// TwinCAT 3 PLC project PRG_B_MachineControl
// Title: B_MachineControl
// Company: RafalOS
// Author: Rafał Osajda
// ProjectVersion: 0.0.0.1
// ProgramVersion: 3.1.4024.0
// libraries:
//   B_Base, * (RafalOS)
//   B_IO, * (RafalOS)
//   Tc2_Standard, * (Beckhoff Automation GmbH)
//   Tc2_System, * (Beckhoff Automation GmbH)
//   Tc3_Module, * (Beckhoff Automation GmbH)
// project tree:
//   DUTs/ ST_Safety.TcDUT, ST_SafetyGroupStates.TcDUT
//   GVLs/ GVL_MCIO.TcGVL, GVL_MCConstans.TcGVL
//   / PlcTask.TcTTO
//   POUs Compilation/ PRG_Compilation.TcPOU
//   POUs/01_MachineControl/ FB_MachineControl.TcPOU
// real-time tasks:
//   TASK PlcTask: cycle T#10ms, priority 20, ADS port 350

CONFIGURATION PRG_B_MachineControl
    RESOURCE PLC ON TwinCAT3
        TASK PlcTask(INTERVAL := T#10ms, PRIORITY := 20);
        PROGRAM PRG_Compilation WITH PlcTask : PRG_Compilation;
    END_RESOURCE
END_CONFIGURATION

// ---- DUTs/ST_Safety.TcDUT
TYPE ST_Safety :
STRUCT
(*	Dane dla programu i podlementów *)	
	flSS1					: FB_BaseFlag;
	flSTO					: FB_BaseFlag;
	flGrzybCh1a				: FB_BaseFlag;
	flGrzybCh1b				: FB_BaseFlag;
(*		*)
	bArmCommand				: BOOL; 	//rozkaz uzbrojenia systemu safety
	// Zmienne bezpieczeństwa globalne
	bRunStop		AT%Q*	: BOOL := TRUE;
	bErrAck			AT%Q*	: BOOL;
	// Zmienne dla grupy 1 - grzyb
	stGroupStates1			: ST_SafetyGroupStates;

END_STRUCT
END_TYPE

// ---- DUTs/ST_SafetyGroupStates.TcDUT
TYPE ST_SafetyGroupStates :
STRUCT
	bInRun			AT%I*	: BOOL;		// grupa działa
	bFbError		AT%I*	: BOOL;		// bład w którymś z FB
	bComError		AT%I*	: BOOL;		// błąd sprzętu
	bOthError		AT%I*	: BOOL;		// inny błąd

	bSS1			AT%I*	: BOOL;		// TRUE - Zgoda na prace jak przechodzi w false zatrzymać napędy
	bSTO			AT%I*	: BOOL;		// TRUE - podawanie zasilania jak przechodzi w false zasilanie odcinane
//	bSS1DlaPRG				: BOOL;		// TRUE - Zgoda na prace jak przechodzi w false zatrzymać napędy
//	bSTODlaPRG				: BOOL;		// TRUE - podawanie zasilania jak przechodzi w false zasilanie odcinane

	bFB_Reset		AT%Q*	: BOOL;
	bL1_EDM			AT%Q*	: BOOL;	
//styki grzyba
	bContact1A		AT%I*	: BOOL;
	bContact1B		AT%I*	: BOOL;
END_STRUCT
END_TYPE

// ---- GVLs/GVL_MCIO.TcGVL
{attribute 'global_init_slot' := '40400'}
{attribute 'qualified_only'}
VAR_GLOBAL
(*	
//Przyciski zmaiany stanu	
	fbprUndefined			: FB_SITP_PolecenieZmianyStanu (ePolecenie := E_SITP_PolecenieZmianyStanu.brak);
	fbprAbort				: FB_SITP_PolecenieZmianyStanu (ePolecenie := E_SITP_PolecenieZmianyStanu.Abort);
   	fbprClear				: FB_SITP_PolecenieZmianyStanu (ePolecenie := E_SITP_PolecenieZmianyStanu.Clear);
    fbprReset				: FB_SITP_PolecenieZmianyStanu (ePolecenie := E_SITP_PolecenieZmianyStanu.Reset);
    fbprStart				: FB_SITP_PolecenieZmianyStanu (ePolecenie := E_SITP_PolecenieZmianyStanu.Start);
    fbprStop				: FB_SITP_PolecenieZmianyStanu (ePolecenie := E_SITP_PolecenieZmianyStanu.Stop);
    fbprHold				: FB_SITP_PolecenieZmianyStanu (ePolecenie := E_SITP_PolecenieZmianyStanu.Hold);
    fbprUnhold				: FB_SITP_PolecenieZmianyStanu (ePolecenie := E_SITP_PolecenieZmianyStanu.Unhold);
    fbprSuspend				: FB_SITP_PolecenieZmianyStanu (ePolecenie := E_SITP_PolecenieZmianyStanu.Suspend);
    fbprUnsuspend			: FB_SITP_PolecenieZmianyStanu (ePolecenie := E_SITP_PolecenieZmianyStanu.Unsuspend);
    fbprComplete			: FB_SITP_PolecenieZmianyStanu (ePolecenie := E_SITP_PolecenieZmianyStanu.Complete);
//przyciski zmiany trybu
	fbprNiedozwolony		: FB_SITP_PolecenieZmianyTrybu (ePolecenie := E_SITP_PolecenieZmianyTrybu.brak);     
	fbprProdukcja			: FB_SITP_PolecenieZmianyTrybu (ePolecenie := E_SITP_PolecenieZmianyTrybu.Produkcja);   
    fbprKonserwacja			: FB_SITP_PolecenieZmianyTrybu (ePolecenie := E_SITP_PolecenieZmianyTrybu.Konserwacja); 
    fbprReczny				: FB_SITP_PolecenieZmianyTrybu (ePolecenie := E_SITP_PolecenieZmianyTrybu.Reczny);      
    fbprMycie				: FB_SITP_PolecenieZmianyTrybu (ePolecenie := E_SITP_PolecenieZmianyTrybu.Mycie);       
    fbprDiagnostyka			: FB_SITP_PolecenieZmianyTrybu (ePolecenie := E_SITP_PolecenieZmianyTrybu.Diagnostyka);
//    fbprUzytkownika2		: FB_SITP_PolecenieZmianyTrybu (ePolecenie := E_SITP_PolecenieZmianyTrybu.Uzytkownika2);
//    fbprUzytkownika3		: FB_SITP_PolecenieZmianyTrybu (ePolecenie := E_SITP_PolecenieZmianyTrybu.Uzytkownika3);
//    fbprUzytkownika4		: FB_SITP_PolecenieZmianyTrybu (ePolecenie := E_SITP_PolecenieZmianyTrybu.Uzytkownika4);
//    fbprUzytkownika5		: FB_SITP_PolecenieZmianyTrybu (ePolecenie := E_SITP_PolecenieZmianyTrybu.Uzytkownika5);
	
//Lampki wieży sygnalizacyjnej
	fbLWiezaCzerwona		: B_IO.FB_LampkaRozszerzona;
	fbLWiezaZolta			: B_IO.FB_LampkaRozszerzona;
	fbLWiezaZielona			: B_IO.FB_LampkaRozszerzona;
	fbLWiezaBiala			: B_IO.FB_LampkaRozszerzona;
	fbLWiezaNiebieska		: B_IO.FB_LampkaRozszerzona;
	
//lampki przycisków polecenia zmiany stanu
	fblprzReset    			: B_IO.FB_LampkaRozszerzona;
    fblprzStart    			: B_IO.FB_LampkaRozszerzona;
    fblprzStop     			: B_IO.FB_LampkaRozszerzona;
    fblprzHold     			: B_IO.FB_LampkaRozszerzona;
    fblprzUnhold   			: B_IO.FB_LampkaRozszerzona;
    fblprzSuspend  			: B_IO.FB_LampkaRozszerzona;
    fblprzUnsuspend			: B_IO.FB_LampkaRozszerzona;
    fblprzAbort    			: B_IO.FB_LampkaRozszerzona;
    fblprzClear    			: B_IO.FB_LampkaRozszerzona;
    fblprzComplete			: B_IO.FB_LampkaRozszerzona;
*)	
END_VAR

// ---- GVLs/GVL_MCConstans.TcGVL
{attribute 'qualified_only'}
VAR_GLOBAL CONSTANT
	
	COUNT_MACHINE_STATES		: INT := 17;	//liczba stanów pracy - max
	COUNT_OPERATION_MODES		: INT := 9;		//liczba trybów pracy - max
	COUNT_STATE_COMMANDS		: INT := 10;	//ilosc polecen zmiany stanu pracy - stany oczekujące np aborted stopped idle itp
	COUNT_MODE_COMMANDS			: INT := 5;		//ilosc polecen zmiany tryby = ilosc trybów pracy
	COUNT_SIGNAL_LAMPS			: INT := 15;
	
//MENU
	MAX_NUMBER_OF_MENU_BUTTONS	: INT := 20;	//max liczba przycisków menu 
END_VAR

// ---- POUs Compilation/PRG_Compilation.TcPOU
PROGRAM PRG_Compilation
VAR
//A01_Element
	fbSITPElement			: FB_SITP_Element;
//A02_EkementStany
	fbStanAborted			: FB_Stan_Aborted;
	fbStanAborting			: FB_Stan_Aborting;
	fbStanClearing			: FB_Stan_Clearing;
	fbStanComplete			: FB_Stan_Complete;
	fbStanCompleting		: FB_Stan_Completing;
	fbStanExecute			: FB_Stan_Execute;
	fbStanHeld				: FB_Stan_Held;
	fbStanHolding			: FB_Stan_Holding;
	fbStanIdle				: FB_Stan_Idle;
	fbStanResseting			: FB_Stan_Resetting;
	fbStanStarting			: FB_Stan_Starting;
	fbStanStopped			: FB_Stan_Stopped;
	fbStanStopping			: FB_Stan_Stopping;
	fbStanSuspended			: FB_Stan_Suspended;
	fbStanSuspending		: FB_Stan_Suspending;
	fbStanUndefined			: FB_Stan_Undefined;
	fbStanUnholding			: FB_Stan_Unholding;
	fbStanUnSuspending		: FB_Stan_Unsuspending;
//A03_ElementTryby
	fbTryb					: FB_Tryb_Uniwersalny;
//04_PolecenieZmiany
	fbPolecenieZmianyStanu			: FB_SITP_PolecenieZmianyStanu (ePolecenie := E_SITP_PolecenieZmianyStanu.Abort);
	fbPolecenieZmianyTrybu			: FB_SITP_PolecenieZmianyTrybu (ePolecenie := E_SITP_PolecenieZmianyTrybu.Produkcja);
//05_SygnalizacjaStanu
	fbSygnalziacjaStanu				: FB_SITP_SygnalizacjaStanu;
//A06_SygnalizacjaStanuStany
	fbSygnalizacjaStanu_Aborted			: FB_SITP_SygnalizacjaStanu_Aborted;
	fbSygnalizacjaStanu_Aborting		: FB_SITP_SygnalizacjaStanu_Aborting;
	fbSygnalizacjaStanu_Clearing		: FB_SITP_SygnalizacjaStanu_Clearing;
	fbSygnalizacjaStanu_Complete		: FB_SITP_SygnalizacjaStanu_Complete;
	fbSygnalizacjaStanu_Completing		: FB_SITP_SygnalizacjaStanu_Completing;
	fbSygnalizacjaStanu_Execute			: FB_SITP_SygnalizacjaStanu_Execute;
	fbSygnalizacjaStanu_Held			: FB_SITP_SygnalizacjaStanu_Held;
	fbSygnalizacjaStanu_Holding			: FB_SITP_SygnalizacjaStanu_Holding;
	fbSygnalizacjaStanu_Idle			: FB_SITP_SygnalizacjaStanu_Idle;
	fbSygnalizacjaStanu_Resseting		: FB_SITP_SygnalizacjaStanu_Resetting;
	fbSygnalizacjaStanu_Starting		: FB_SITP_SygnalizacjaStanu_Starting;
	fbSygnalizacjaStanu_Stopped			: FB_SITP_SygnalizacjaStanu_Stopped;
	fbSygnalizacjaStanu_Stopping		: FB_SITP_SygnalizacjaStanu_Stopping;
	fbSygnalizacjaStanu_Suspended		: FB_SITP_SygnalizacjaStanu_Suspended;
	fbSygnalizacjaStanu_Suspending		: FB_SITP_SygnalizacjaStanu_Suspending;
	fbSygnalizacjaStanu_Undefined		: FB_SITP_SygnalizacjaStanu_Undefined;
	fbSygnalizacjaStanu_Unholding		: FB_SITP_SygnalizacjaStanu_Unholding;
	fbSygnalizacjaStanu_UnSuspending	: FB_SITP_SygnalizacjaStanu_Unsuspending;	
//A10_SITP
	stSafety						: ST_Safety;
//SPM
	fbSPM							: FB_SPM;

	
END_VAR

END_PROGRAM

// ---- POUs/01_MachineControl/FB_MachineControl.TcPOU
FUNCTION_BLOCK FB_MachineControl EXTENDS FB_BaseTopElement
VAR

END_VAR

END_FUNCTION_BLOCK
